// TIA Portal V18 export
DATA_BLOCK "Process_DB"   // DB1
VERSION : 0.1
// stored: Access Unpublished, AutoNumber true, DBAccessibleFromOPCUA true, DBAccessibleFromWebserver true, InstanceOfName Coagulation.Process, InstanceOfType FB, Namespace Coagulation
"Coagulation.Process"
BEGIN
END_DATA_BLOCK
